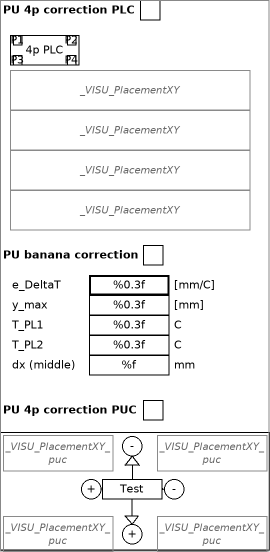
VISUALIZATION _VISU_FineAlignment  // 270x552
VAR_IN_OUT
	mInst : FB_FineAlignement;
END_VAR
    Rectangle (0,432 270x118)
    Rectangle (0,0 259x427)
    Rectangle (0,0 140x20), "PU 4p correction PLC"
    RoundedRectangle (140,0 20x20)
        toggle mInst._bEnable_4p
    Rectangle (0,245 140x20), "PU banana correction"
    RoundedRectangle (143,245 20x20)
        toggle mInst._bEnable_banana
    Rectangle (0,400 140x20), "PU 4p correction PUC"
    RoundedRectangle (143,400 20x20)
        toggle mInst._bEnablePuc_4p
    Frame (10,70 240x40)
        shows _VISU_PlacementXY(m_Inst := mInst._fbPlcCorrPoints[1])
    Group (10,35 69x30)
        RoundedRectangle (0,0 69x30), "4p PLC"
        Rectangle (3,0 9x10), "P1"
        Rectangle (57,0 9x10), "P2"
        Rectangle (57,20 9x10), "P4"
        Rectangle (3,20 9x10), "P3"
    Frame (10,110 240x40)
        shows _VISU_PlacementXY(m_Inst := mInst._fbPlcCorrPoints[2])
    Frame (10,150 240x40)
        shows _VISU_PlacementXY(m_Inst := mInst._fbPlcCorrPoints[3])
    Frame (10,190 240x40)
        shows _VISU_PlacementXY(m_Inst := mInst._fbPlcCorrPoints[4])
    Rectangle (89,275 80x20), "%0.3f", text variable: mInst._e_max_per_deltaT
        OnMouseClick: write the text variable via Default
    Rectangle (89,295 80x20), "%0.3f", text variable: mInst._y_max
    Rectangle (9,275 80x20), "e_DeltaT"
    Rectangle (9,295 80x20), "y_max"
    Rectangle (171,295 51x20), "[mm]"
    Rectangle (171,275 51x20), "[mm/C]"
    Rectangle (89,315 80x20), "%0.3f", text variable: mInst._fT1
    Rectangle (89,335 80x20), "%0.3f", text variable: mInst._fT2
    Rectangle (9,315 80x20), "T_PL1"
    Rectangle (9,335 80x20), "T_PL2"
    Rectangle (171,315 51x20), "C"
    Rectangle (171,335 51x20), "C"
    Rectangle (89,355 80x20), "%f", text variable: mInst._dx_middle
    Rectangle (9,355 80x20), "dx (middle)"
    Rectangle (171,355 51x20), "mm"
    Frame (3,435 110x36)
        shows _VISU_PlacementXY_puc(mInst := mInst._pAdsCam^.stAds.sI_CorrectionPointIndication[1], aName := mInst.aPucPointNames[1], bSelected := mInst.bSelected[1], bSelect := mInst.bSelect[1])
    Frame (157,435 110x36)
        shows _VISU_PlacementXY_puc(mInst := mInst._pAdsCam^.stAds.sI_CorrectionPointIndication[2], aName := mInst.aPucPointNames[2], bSelected := mInst.bSelected[2], bSelect := mInst.bSelect[2])
    Frame (3,516 110x36)
        shows _VISU_PlacementXY_puc(mInst := mInst._pAdsCam^.stAds.sI_CorrectionPointIndication[3], aName := mInst.aPucPointNames[3], bSelected := mInst.bSelected[3], bSelect := mInst.bSelect[3])
    Frame (157,516 110x36)
        shows _VISU_PlacementXY_puc(mInst := mInst._pAdsCam^.stAds.sI_CorrectionPointIndication[4], aName := mInst.aPucPointNames[4], bSelected := mInst.bSelected[4], bSelect := mInst.bSelect[4])
    Group (81,436 103x108), invisible if: NOT mInst._bUT_4pPuc
        Ellipse (41,0 20x20), "-"
            toggle mInst.bYMinus
        Ellipse (41,88 20x20), "+"
            toggle mInst.bYPlus
        Polyline (51,29) (44,29) (51,20) (58,29) (51,29) (51,46)
        Polyline (51,80) (44,80) (51,88) (57,80) (51,80) (51,63)
        Ellipse (83,43 20x20), "-"
            toggle mInst.bXMinus
        Ellipse (0,43 20x20), "+"
            toggle mInst.bXPlus
        Polyline (28,53) (28,47) (21,53) (28,59) (28,53) (44,53)
        Polyline (74,54) (74,46) (82,53) (74,59) (74,53) (58,53)
        Rectangle (41,43 20x20), "P%d", text variable: mInst.nSelectedPoint
    RoundedRectangle (102,479 60x20), "Test", invisible if: mInst._bUT_4pPuc
        toggle mInst._bUT_4pPuc
END_VISUALIZATION

(* stored: Version 1.1.0.1, ProductVersion 3.1.4024.11
   Visu _VISU_FineAlignment: Id {bf481098-27ac-4095-a5ca-73b74d9effd8} *)
